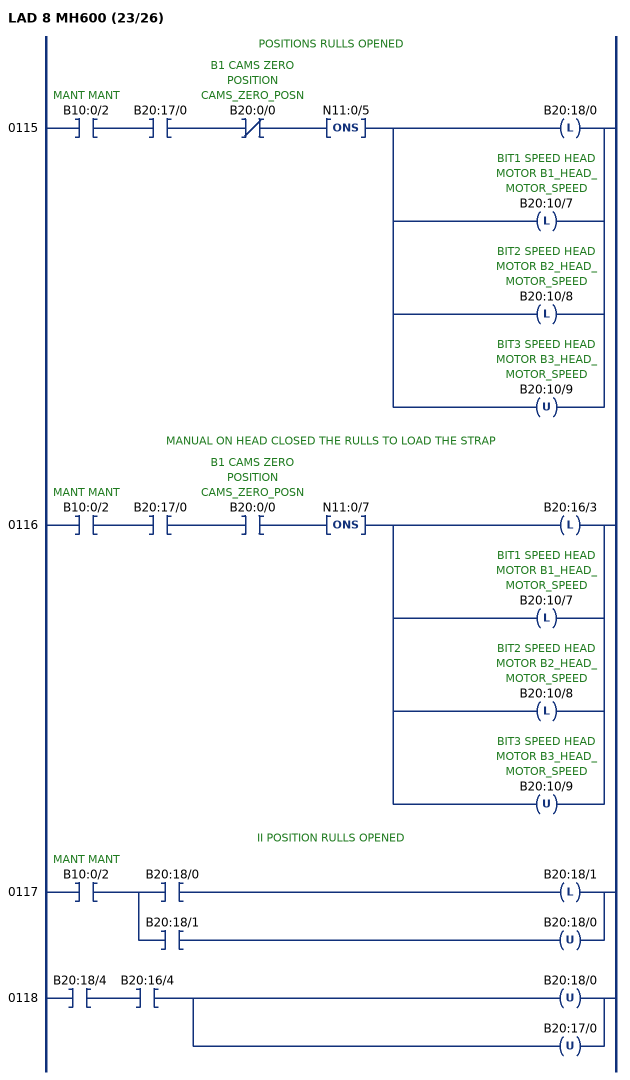
% Rung: 115 %
% POSITIONS RULLS OPENED %
SOR XIC B10:0/2 XIC B20:17/0 XIO B20:0/0 ONS N11:0/5 BST OTL B20:18/0 NXB BST OTL B20:10/7 NXB BST OTL B20:10/8 NXB OTU B20:10/9 BND BND BND EOR
%   B10:0/2  MANT  "MANT" %
%   B20:0/0  CAMS_ZERO_POSN  "B1 CAMS ZERO POSITION" %
%   B20:10/7  B1_HEAD_MOTOR_SPEED  "BIT1 SPEED HEAD MOTOR" %
%   B20:10/8  B2_HEAD_MOTOR_SPEED  "BIT2 SPEED HEAD MOTOR" %
%   B20:10/9  B3_HEAD_MOTOR_SPEED  "BIT3 SPEED HEAD MOTOR" %
% Rung: 116 %
% MANUAL ON HEAD CLOSED THE RULLS TO LOAD THE STRAP %
SOR XIC B10:0/2 XIC B20:17/0 XIC B20:0/0 ONS N11:0/7 BST OTL B20:16/3 NXB BST OTL B20:10/7 NXB BST OTL B20:10/8 NXB OTU B20:10/9 BND BND BND EOR
%   B10:0/2  MANT  "MANT" %
%   B20:0/0  CAMS_ZERO_POSN  "B1 CAMS ZERO POSITION" %
%   B20:10/7  B1_HEAD_MOTOR_SPEED  "BIT1 SPEED HEAD MOTOR" %
%   B20:10/8  B2_HEAD_MOTOR_SPEED  "BIT2 SPEED HEAD MOTOR" %
%   B20:10/9  B3_HEAD_MOTOR_SPEED  "BIT3 SPEED HEAD MOTOR" %
% Rung: 117 %
% II POSITION RULLS OPENED %
SOR XIC B10:0/2 BST XIC B20:18/0 OTL B20:18/1 NXB XIC B20:18/1 OTU B20:18/0 BND EOR
%   B10:0/2  MANT  "MANT" %
% Rung: 118 %
SOR XIC B20:18/4 XIC B20:16/4 BST OTU B20:18/0 NXB OTU B20:17/0 BND EOR

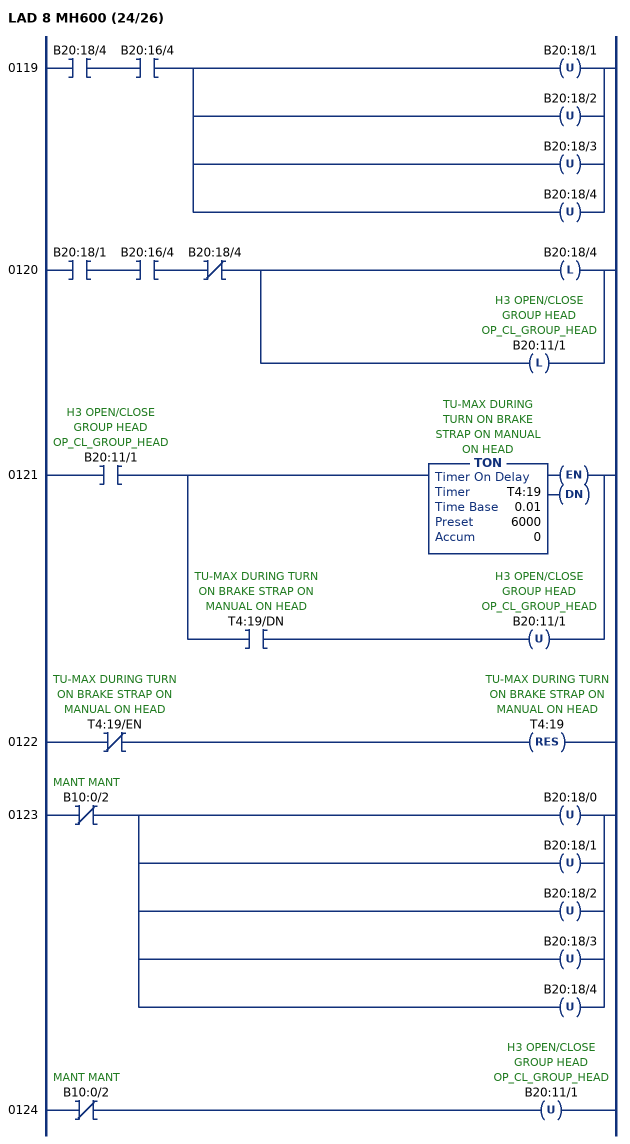
% Rung: 119 %
SOR XIC B20:18/4 XIC B20:16/4 BST OTU B20:18/1 NXB BST OTU B20:18/2 NXB BST OTU B20:18/3 NXB OTU B20:18/4 BND BND BND EOR
% Rung: 120 %
SOR XIC B20:18/1 XIC B20:16/4 XIO B20:18/4 BST OTL B20:18/4 NXB OTL B20:11/1 BND EOR
%   B20:11/1  OP_CL_GROUP_HEAD  "H3 OPEN/CLOSE GROUP HEAD" %
% Rung: 121 %
SOR XIC B20:11/1 BST TON T4:19 0.01 6000 0 NXB XIC T4:19/DN OTU B20:11/1 BND EOR
%   B20:11/1  OP_CL_GROUP_HEAD  "H3 OPEN/CLOSE GROUP HEAD" %
%   T4:19  "TU-MAX DURING TURN ON BRAKE STRAP ON MANUAL ON HEAD" %
% Rung: 122 %
SOR XIO T4:19/EN RES T4:19 EOR
%   T4:19  "TU-MAX DURING TURN ON BRAKE STRAP ON MANUAL ON HEAD" %
% Rung: 123 %
SOR XIO B10:0/2 BST OTU B20:18/0 NXB BST OTU B20:18/1 NXB BST OTU B20:18/2 NXB BST OTU B20:18/3 NXB OTU B20:18/4 BND BND BND BND EOR
%   B10:0/2  MANT  "MANT" %
% Rung: 124 %
SOR XIO B10:0/2 OTU B20:11/1 EOR
%   B10:0/2  MANT  "MANT" %
%   B20:11/1  OP_CL_GROUP_HEAD  "H3 OPEN/CLOSE GROUP HEAD" %

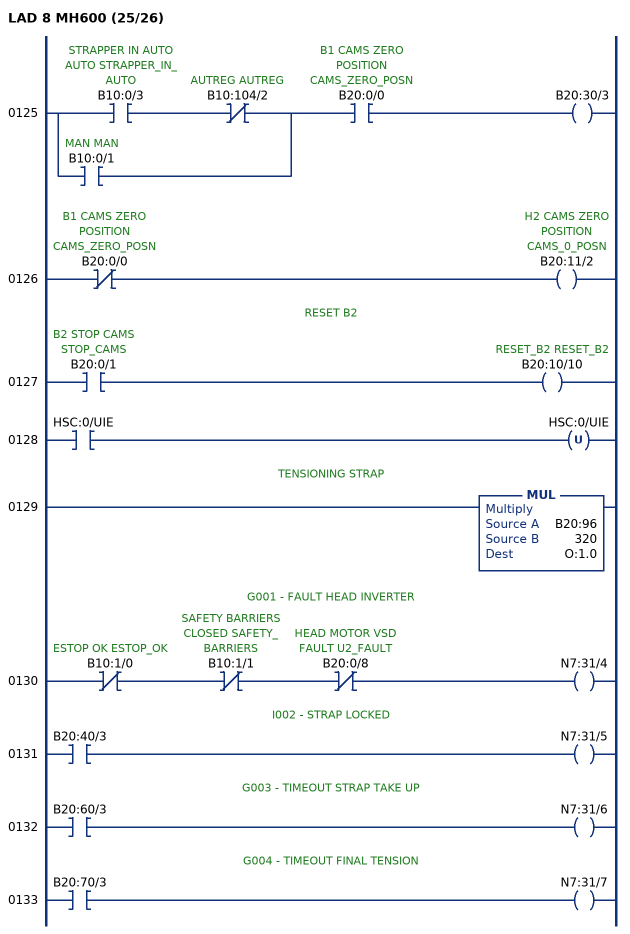
% Rung: 125 %
SOR BST XIC B10:0/3 XIO B10:104/2 NXB XIC B10:0/1 BND XIC B20:0/0 OTE B20:30/3 EOR
%   B10:0/3  STRAPPER_IN_AUTO  "STRAPPER IN AUTO AUTO" %
%   B10:104/2  AUTREG  "AUTREG" %
%   B10:0/1  MAN  "MAN" %
%   B20:0/0  CAMS_ZERO_POSN  "B1 CAMS ZERO POSITION" %
% Rung: 126 %
SOR XIO B20:0/0 OTE B20:11/2 EOR
%   B20:0/0  CAMS_ZERO_POSN  "B1 CAMS ZERO POSITION" %
%   B20:11/2  CAMS_0_POSN  "H2 CAMS ZERO POSITION" %
% Rung: 127 %
% RESET B2 %
SOR XIC B20:0/1 OTE B20:10/10 EOR
%   B20:0/1  STOP_CAMS  "B2 STOP CAMS" %
%   B20:10/10  RESET_B2  "RESET_B2" %
% Rung: 128 %
SOR XIC HSC:0/UIE OTU HSC:0/UIE EOR
% Rung: 129 %
% TENSIONING STRAP %
SOR MUL B20:96 320 O:1.0 EOR
% Rung: 130 %
% G001 - FAULT HEAD INVERTER %
SOR XIO B10:1/0 XIO B10:1/1 XIO B20:0/8 OTE N7:31/4 EOR
%   B10:1/0  ESTOP_OK  "ESTOP OK" %
%   B10:1/1  SAFETY_BARRIERS  "SAFETY BARRIERS CLOSED" %
%   B20:0/8  U2_FAULT  "HEAD MOTOR VSD FAULT" %
% Rung: 131 %
% I002 - STRAP LOCKED %
SOR XIC B20:40/3 OTE N7:31/5 EOR
% Rung: 132 %
% G003 - TIMEOUT STRAP TAKE UP %
SOR XIC B20:60/3 OTE N7:31/6 EOR
% Rung: 133 %
% G004 - TIMEOUT FINAL TENSION %
SOR XIC B20:70/3 OTE N7:31/7 EOR

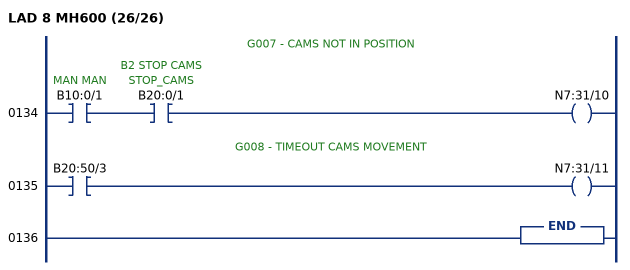
% Rung: 134 %
% G007 - CAMS NOT IN POSITION %
SOR XIC B10:0/1 XIC B20:0/1 OTE N7:31/10 EOR
%   B10:0/1  MAN  "MAN" %
%   B20:0/1  STOP_CAMS  "B2 STOP CAMS" %
% Rung: 135 %
% G008 - TIMEOUT CAMS MOVEMENT %
SOR XIC B20:50/3 OTE N7:31/11 EOR
% Rung: 136 %
SOR END EOR

LADDER 9 "ORGANIT."
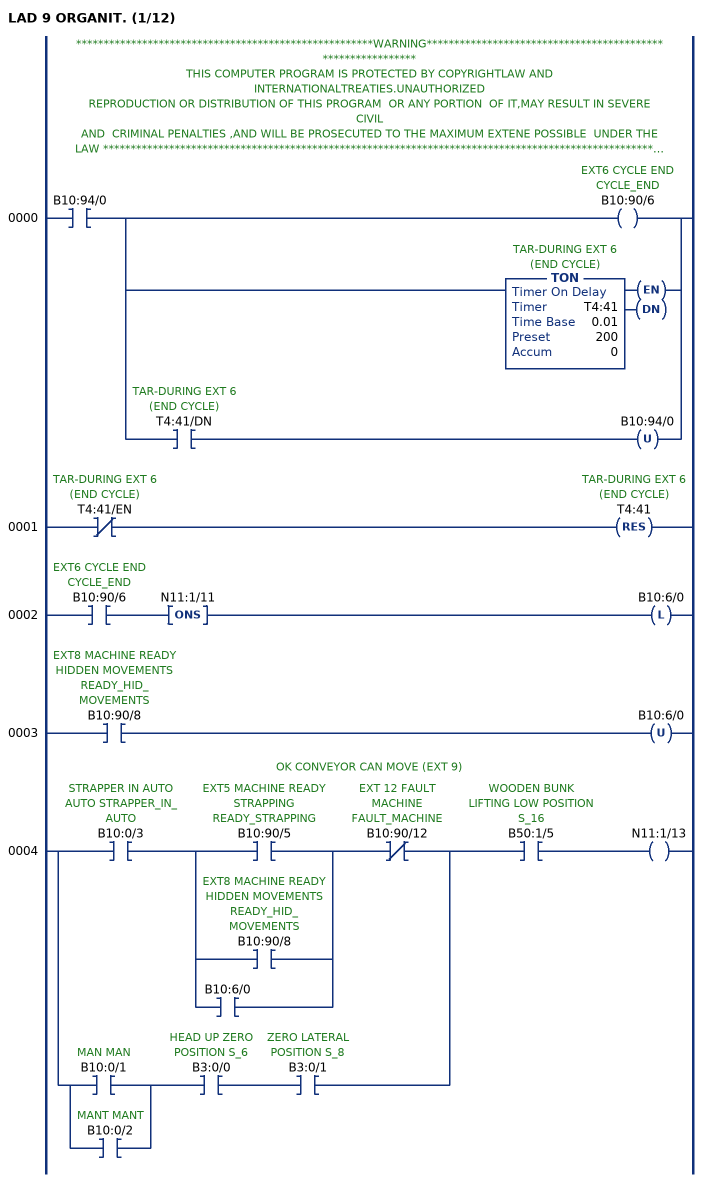
% Rung: 0 %
% ******************************************************WARNING************************************************************
% THIS COMPUTER PROGRAM IS PROTECTED BY COPYRIGHTLAW AND  INTERNATIONALTREATIES.UNAUTHORIZED
%  REPRODUCTION OR DISTRIBUTION OF THIS PROGRAM  OR ANY PORTION  OF IT,MAY RESULT IN SEVERE CIVIL
% AND  CRIMINAL PENALTIES ,AND WILL BE PROSECUTED TO THE MAXIMUM EXTENE POSSIBLE  UNDER THE LAW **************************************************************************************************************************
% INTERFACE SIGNALS - CYCLE END %
SOR XIC B10:94/0 BST OTE B10:90/6 NXB BST TON T4:41 0.01 200 0 NXB XIC T4:41/DN OTU B10:94/0 BND BND EOR
%   B10:90/6  CYCLE_END  "EXT6 CYCLE END" %
%   T4:41  "TAR-DURING EXT 6 (END CYCLE)" %
% Rung: 1 %
SOR XIO T4:41/EN RES T4:41 EOR
%   T4:41  "TAR-DURING EXT 6 (END CYCLE)" %
% Rung: 2 %
SOR XIC B10:90/6 ONS N11:1/11 OTL B10:6/0 EOR
%   B10:90/6  CYCLE_END  "EXT6 CYCLE END" %
% Rung: 3 %
SOR XIC B10:90/8 OTU B10:6/0 EOR
%   B10:90/8  READY_HID_MOVEMENTS  "EXT8 MACHINE READY HIDDEN MOVEMENTS" %
% Rung: 4 %
% OK CONVEYOR CAN MOVE (EXT 9) %
SOR BST XIC B10:0/3 BST XIC B10:90/5 NXB BST XIC B10:90/8 NXB XIC B10:6/0 BND BND XIO B10:90/12 NXB BST XIC B10:0/1 NXB XIC B10:0/2 BND XIC B3:0/0 XIC B3:0/1 BND XIC B50:1/5 OTE N11:1/13 EOR
%   B10:0/3  STRAPPER_IN_AUTO  "STRAPPER IN AUTO AUTO" %
%   B10:90/5  READY_STRAPPING  "EXT5 MACHINE READY STRAPPING" %
%   B10:90/8  READY_HID_MOVEMENTS  "EXT8 MACHINE READY HIDDEN MOVEMENTS" %
%   B10:90/12  FAULT_MACHINE  "EXT 12 FAULT MACHINE" %
%   B10:0/1  MAN  "MAN" %
%   B10:0/2  MANT  "MANT" %
%   B3:0/0  S_6  "HEAD UP ZERO POSITION" %
%   B3:0/1  S_8  "ZERO LATERAL POSITION" %
%   B50:1/5  S_16  "WOODEN BUNK LIFTING LOW POSITION" %

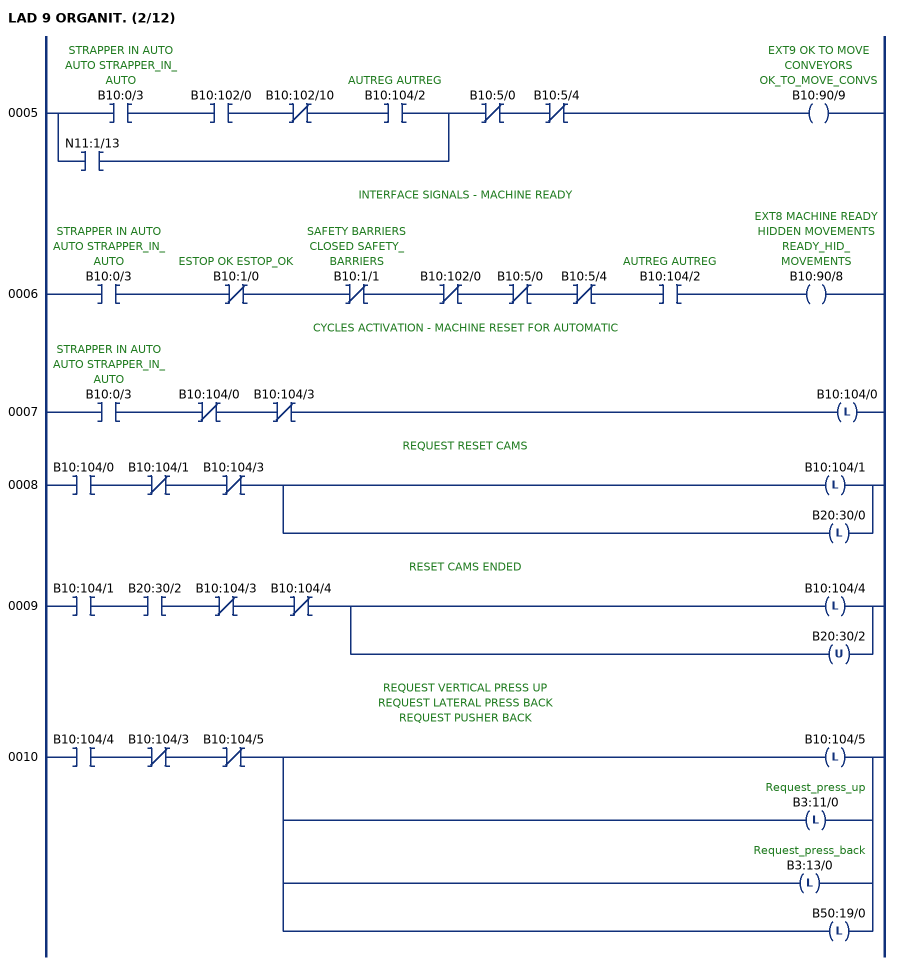
% Rung: 5 %
SOR BST XIC B10:0/3 XIC B10:102/0 XIO B10:102/10 XIC B10:104/2 NXB XIC N11:1/13 BND XIO B10:5/0 XIO B10:5/4 OTE B10:90/9 EOR
%   B10:0/3  STRAPPER_IN_AUTO  "STRAPPER IN AUTO AUTO" %
%   B10:104/2  AUTREG  "AUTREG" %
%   B10:90/9  OK_TO_MOVE_CONVS  "EXT9 OK TO MOVE CONVEYORS" %
% Rung: 6 %
% INTERFACE SIGNALS - MACHINE READY %
SOR XIC B10:0/3 XIO B10:1/0 XIO B10:1/1 XIO B10:102/0 XIO B10:5/0 XIO B10:5/4 XIC B10:104/2 OTE B10:90/8 EOR
%   B10:0/3  STRAPPER_IN_AUTO  "STRAPPER IN AUTO AUTO" %
%   B10:1/0  ESTOP_OK  "ESTOP OK" %
%   B10:1/1  SAFETY_BARRIERS  "SAFETY BARRIERS CLOSED" %
%   B10:104/2  AUTREG  "AUTREG" %
%   B10:90/8  READY_HID_MOVEMENTS  "EXT8 MACHINE READY HIDDEN MOVEMENTS" %
% Rung: 7 %
% CYCLES ACTIVATION - MACHINE RESET FOR AUTOMATIC %
SOR XIC B10:0/3 XIO B10:104/0 XIO B10:104/3 OTL B10:104/0 EOR
%   B10:0/3  STRAPPER_IN_AUTO  "STRAPPER IN AUTO AUTO" %
% Rung: 8 %
% REQUEST RESET CAMS %
SOR XIC B10:104/0 XIO B10:104/1 XIO B10:104/3 BST OTL B10:104/1 NXB OTL B20:30/0 BND EOR
% Rung: 9 %
% RESET CAMS ENDED %
SOR XIC B10:104/1 XIC B20:30/2 XIO B10:104/3 XIO B10:104/4 BST OTL B10:104/4 NXB OTU B20:30/2 BND EOR
% Rung: 10 %
% REQUEST VERTICAL PRESS UP
% REQUEST LATERAL PRESS BACK
% REQUEST PUSHER BACK %
SOR XIC B10:104/4 XIO B10:104/3 XIO B10:104/5 BST OTL B10:104/5 NXB BST OTL B3:11/0 NXB BST OTL B3:13/0 NXB OTL B50:19/0 BND BND BND EOR
%   B3:11/0  "Request_press_up" %
%   B3:13/0  "Request_press_back" %

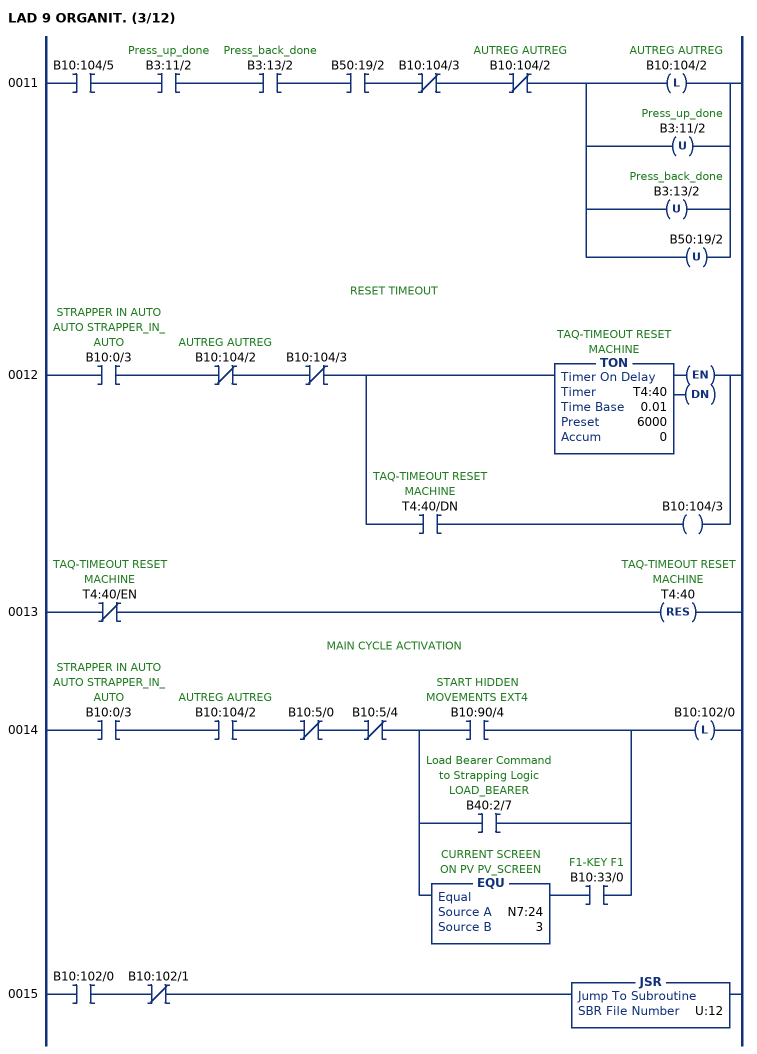
% Rung: 11 %
SOR XIC B10:104/5 XIC B3:11/2 XIC B3:13/2 XIC B50:19/2 XIO B10:104/3 XIO B10:104/2 BST OTL B10:104/2 NXB BST BST OTU B3:11/2 NXB OTU B3:13/2 BND NXB OTU B50:19/2 BND BND EOR
%   B3:11/2  "Press_up_done" %
%   B3:13/2  "Press_back_done" %
%   B10:104/2  AUTREG  "AUTREG" %
% Rung: 12 %
% RESET TIMEOUT %
SOR XIC B10:0/3 XIO B10:104/2 XIO B10:104/3 BST TON T4:40 0.01 6000 0 NXB XIC T4:40/DN OTE B10:104/3 BND EOR
%   B10:0/3  STRAPPER_IN_AUTO  "STRAPPER IN AUTO AUTO" %
%   B10:104/2  AUTREG  "AUTREG" %
%   T4:40  "TAQ-TIMEOUT RESET MACHINE" %
% Rung: 13 %
SOR XIO T4:40/EN RES T4:40 EOR
%   T4:40  "TAQ-TIMEOUT RESET MACHINE" %
% Rung: 14 %
% MAIN CYCLE ACTIVATION %
SOR XIC B10:0/3 XIC B10:104/2 XIO B10:5/0 XIO B10:5/4 BST XIC B10:90/4 NXB XIC B40:2/7 NXB EQU N7:24 3 XIC B10:33/0 BND OTL B10:102/0 EOR
%   B10:0/3  STRAPPER_IN_AUTO  "STRAPPER IN AUTO AUTO" %
%   B10:104/2  AUTREG  "AUTREG" %
%   B10:90/4  EXT4  "START HIDDEN MOVEMENTS" %
%   B40:2/7  LOAD_BEARER  "Load Bearer Command to Strapping Logic" %
%   N7:24  PV_SCREEN  "CURRENT SCREEN ON PV" %
%   B10:33/0  F1  "F1-KEY" %
% Rung: 15 %
SOR XIC B10:102/0 XIO B10:102/1 JSR U:12 EOR

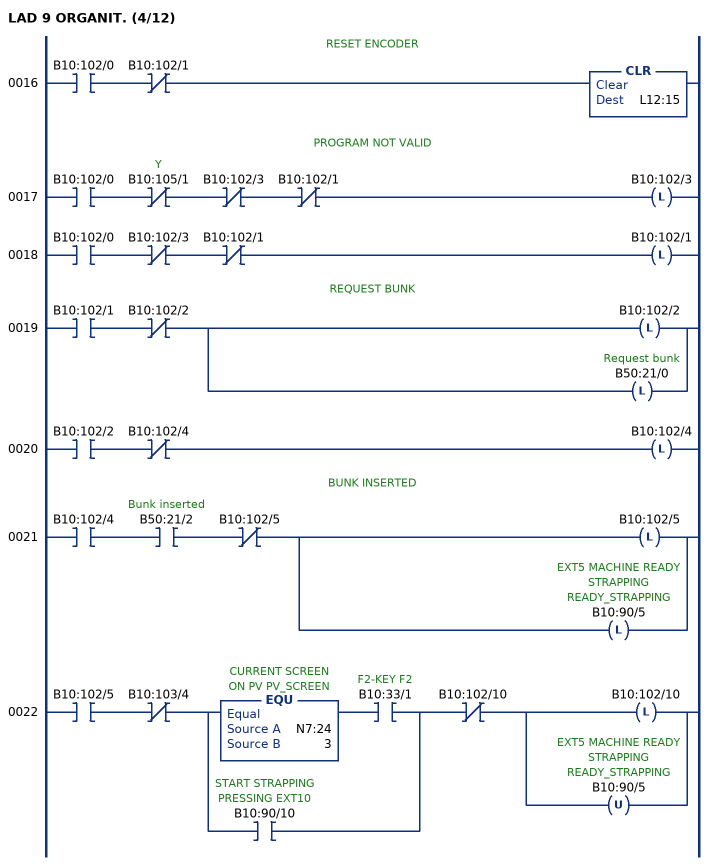
% Rung: 16 %
% RESET ENCODER %
SOR XIC B10:102/0 XIO B10:102/1 CLR L12:15 EOR
% Rung: 17 %
% PROGRAM NOT VALID %
SOR XIC B10:102/0 XIO B10:105/1 XIO B10:102/3 XIO B10:102/1 OTL B10:102/3 EOR
%   B10:105/1  "Y" %
% Rung: 18 %
SOR XIC B10:102/0 XIO B10:102/3 XIO B10:102/1 OTL B10:102/1 EOR
% Rung: 19 %
% REQUEST BUNK %
SOR XIC B10:102/1 XIO B10:102/2 BST OTL B10:102/2 NXB OTL B50:21/0 BND EOR
%   B50:21/0  "Request bunk" %
% Rung: 20 %
SOR XIC B10:102/2 XIO B10:102/4 OTL B10:102/4 EOR
% Rung: 21 %
% BUNK INSERTED %
SOR XIC B10:102/4 XIC B50:21/2 XIO B10:102/5 BST OTL B10:102/5 NXB OTL B10:90/5 BND EOR
%   B50:21/2  "Bunk inserted" %
%   B10:90/5  READY_STRAPPING  "EXT5 MACHINE READY STRAPPING" %
% Rung: 22 %
SOR XIC B10:102/5 XIO B10:103/4 BST EQU N7:24 3 XIC B10:33/1 NXB XIC B10:90/10 BND XIO B10:102/10 BST OTL B10:102/10 NXB OTU B10:90/5 BND EOR
%   N7:24  PV_SCREEN  "CURRENT SCREEN ON PV" %
%   B10:33/1  F2  "F2-KEY" %
%   B10:90/10  EXT10  "START STRAPPING PRESSING" %
%   B10:90/5  READY_STRAPPING  "EXT5 MACHINE READY STRAPPING" %

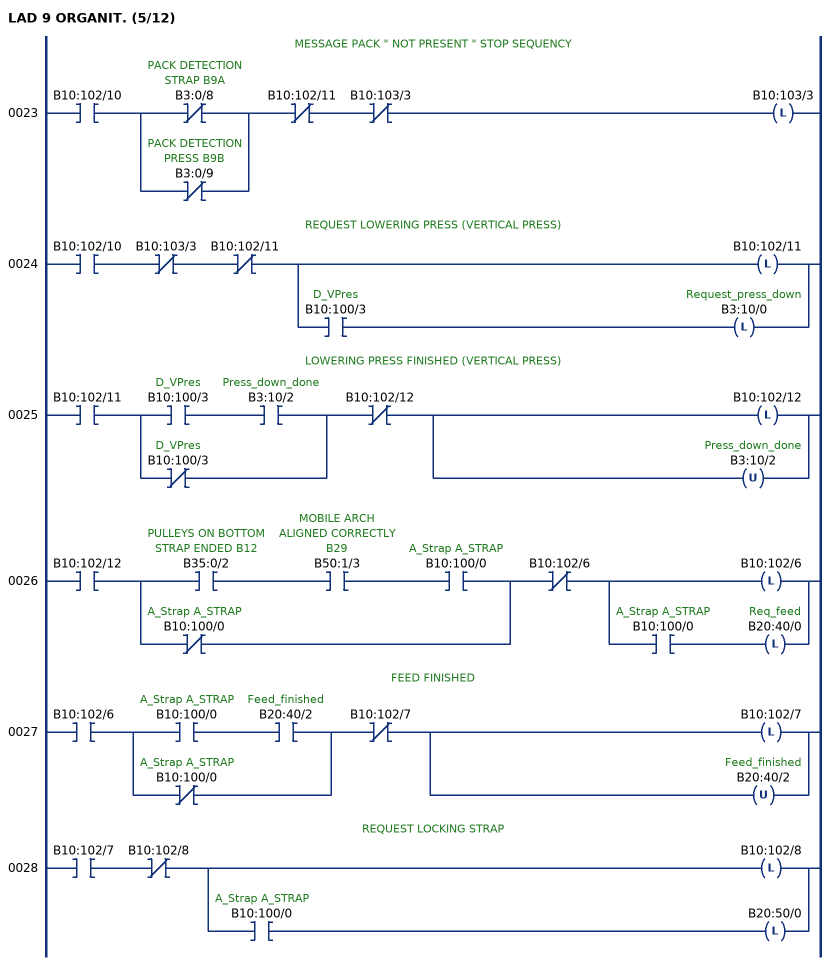
% Rung: 23 %
% MESSAGE PACK " NOT PRESENT " STOP SEQUENCY %
SOR XIC B10:102/10 BST XIO B3:0/8 NXB XIO B3:0/9 BND XIO B10:102/11 XIO B10:103/3 OTL B10:103/3 EOR
%   B3:0/8  B9A  "PACK DETECTION STRAP" %
%   B3:0/9  B9B  "PACK DETECTION PRESS" %
% Rung: 24 %
% REQUEST LOWERING PRESS (VERTICAL PRESS) %
SOR XIC B10:102/10 XIO B10:103/3 XIO B10:102/11 BST OTL B10:102/11 NXB XIC B10:100/3 OTL B3:10/0 BND EOR
%   B10:100/3  "D_VPres" %
%   B3:10/0  "Request_press_down" %
% Rung: 25 %
% LOWERING PRESS FINISHED (VERTICAL PRESS) %
SOR XIC B10:102/11 BST XIC B10:100/3 XIC B3:10/2 NXB XIO B10:100/3 BND XIO B10:102/12 BST OTL B10:102/12 NXB OTU B3:10/2 BND EOR
%   B10:100/3  "D_VPres" %
%   B3:10/2  "Press_down_done" %
% Rung: 26 %
SOR XIC B10:102/12 BST XIC B35:0/2 XIC B50:1/3 XIC B10:100/0 NXB XIO B10:100/0 BND XIO B10:102/6 BST OTL B10:102/6 NXB XIC B10:100/0 OTL B20:40/0 BND EOR
%   B35:0/2  B12  "PULLEYS ON BOTTOM STRAP ENDED" %
%   B50:1/3  B29  "MOBILE ARCH ALIGNED CORRECTLY" %
%   B10:100/0  A_STRAP  "A_Strap" %
%   B20:40/0  "Req_feed" %
% Rung: 27 %
% FEED FINISHED %
SOR XIC B10:102/6 BST XIC B10:100/0 XIC B20:40/2 NXB XIO B10:100/0 BND XIO B10:102/7 BST OTL B10:102/7 NXB OTU B20:40/2 BND EOR
%   B10:100/0  A_STRAP  "A_Strap" %
%   B20:40/2  "Feed_finished" %
% Rung: 28 %
% REQUEST LOCKING STRAP %
SOR XIC B10:102/7 XIO B10:102/8 BST OTL B10:102/8 NXB XIC B10:100/0 OTL B20:50/0 BND EOR
%   B10:100/0  A_STRAP  "A_Strap" %

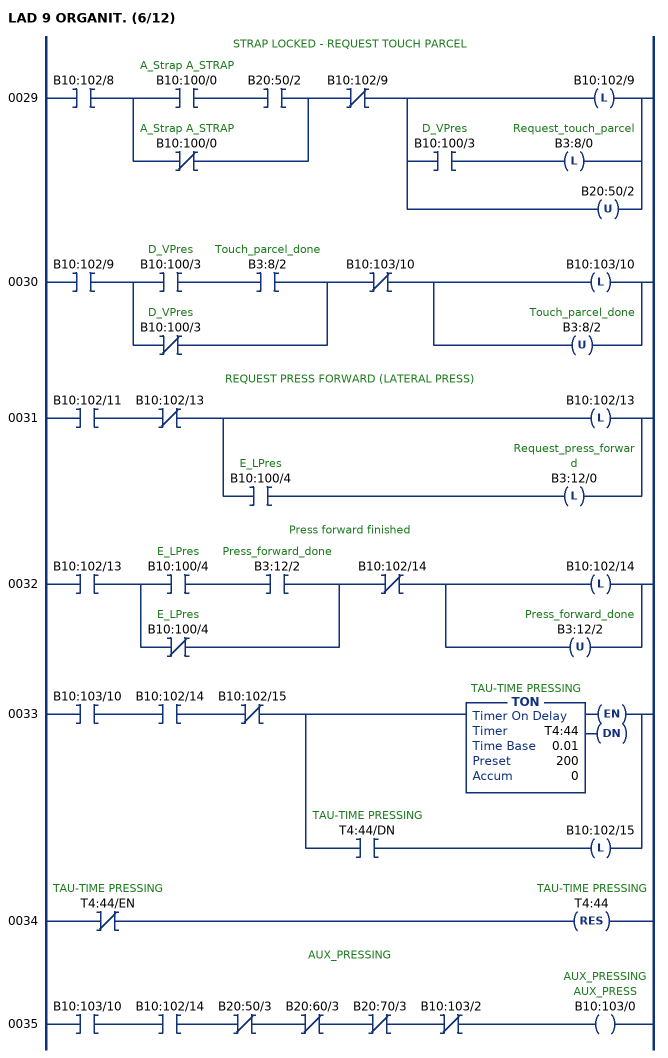
% Rung: 29 %
% STRAP LOCKED - REQUEST TOUCH PARCEL %
SOR XIC B10:102/8 BST XIC B10:100/0 XIC B20:50/2 NXB XIO B10:100/0 BND XIO B10:102/9 BST BST OTL B10:102/9 NXB XIC B10:100/3 OTL B3:8/0 BND NXB OTU B20:50/2 BND EOR
%   B10:100/0  A_STRAP  "A_Strap" %
%   B10:100/3  "D_VPres" %
%   B3:8/0  "Request_touch_parcel" %
% Rung: 30 %
SOR XIC B10:102/9 BST XIC B10:100/3 XIC B3:8/2 NXB XIO B10:100/3 BND XIO B10:103/10 BST OTL B10:103/10 NXB OTU B3:8/2 BND EOR
%   B10:100/3  "D_VPres" %
%   B3:8/2  "Touch_parcel_done" %
% Rung: 31 %
% REQUEST PRESS FORWARD (LATERAL PRESS) %
SOR XIC B10:102/11 XIO B10:102/13 BST OTL B10:102/13 NXB XIC B10:100/4 OTL B3:12/0 BND EOR
%   B10:100/4  "E_LPres" %
%   B3:12/0  "Request_press_forwar d" %
% Rung: 32 %
% Press forward finished %
SOR XIC B10:102/13 BST XIC B10:100/4 XIC B3:12/2 NXB XIO B10:100/4 BND XIO B10:102/14 BST OTL B10:102/14 NXB OTU B3:12/2 BND EOR
%   B10:100/4  "E_LPres" %
%   B3:12/2  "Press_forward_done" %
% Rung: 33 %
SOR XIC B10:103/10 XIC B10:102/14 XIO B10:102/15 BST TON T4:44 0.01 200 0 NXB XIC T4:44/DN OTL B10:102/15 BND EOR
%   T4:44  "TAU-TIME PRESSING" %
% Rung: 34 %
SOR XIO T4:44/EN RES T4:44 EOR
%   T4:44  "TAU-TIME PRESSING" %
% Rung: 35 %
% AUX_PRESSING %
SOR XIC B10:103/10 XIC B10:102/14 XIO B20:50/3 XIO B20:60/3 XIO B20:70/3 XIO B10:103/2 OTE B10:103/0 EOR
%   B10:103/0  AUX_PRESS  "AUX_PRESSING" %

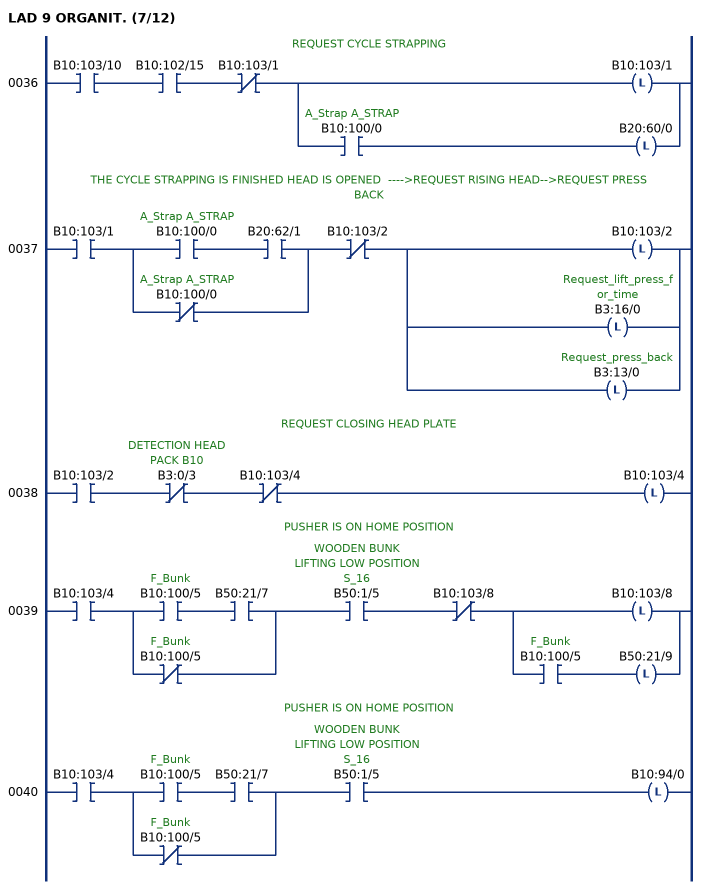
% Rung: 36 %
% REQUEST CYCLE STRAPPING %
SOR XIC B10:103/10 XIC B10:102/15 XIO B10:103/1 BST OTL B10:103/1 NXB XIC B10:100/0 OTL B20:60/0 BND EOR
%   B10:100/0  A_STRAP  "A_Strap" %
% Rung: 37 %
% THE CYCLE STRAPPING IS FINISHED HEAD IS OPENED  ---->REQUEST RISING HEAD-->REQUEST PRESS BACK %
SOR XIC B10:103/1 BST XIC B10:100/0 XIC B20:62/1 NXB XIO B10:100/0 BND XIO B10:103/2 BST OTL B10:103/2 NXB BST OTL B3:16/0 NXB OTL B3:13/0 BND BND EOR
%   B10:100/0  A_STRAP  "A_Strap" %
%   B3:16/0  "Request_lift_press_f or_time" %
%   B3:13/0  "Request_press_back" %
% Rung: 38 %
% REQUEST CLOSING HEAD PLATE %
SOR XIC B10:103/2 XIO B3:0/3 XIO B10:103/4 OTL B10:103/4 EOR
%   B3:0/3  B10  "DETECTION HEAD PACK" %
% Rung: 39 %
% PUSHER IS ON HOME POSITION %
SOR XIC B10:103/4 BST XIC B10:100/5 XIC B50:21/7 NXB XIO B10:100/5 BND XIC B50:1/5 XIO B10:103/8 BST OTL B10:103/8 NXB XIC B10:100/5 OTL B50:21/9 BND EOR
%   B10:100/5  "F_Bunk" %
%   B50:1/5  S_16  "WOODEN BUNK LIFTING LOW POSITION" %
% Rung: 40 %
% PUSHER IS ON HOME POSITION %
SOR XIC B10:103/4 BST XIC B10:100/5 XIC B50:21/7 NXB XIO B10:100/5 BND XIC B50:1/5 OTL B10:94/0 EOR
%   B10:100/5  "F_Bunk" %
%   B50:1/5  S_16  "WOODEN BUNK LIFTING LOW POSITION" %

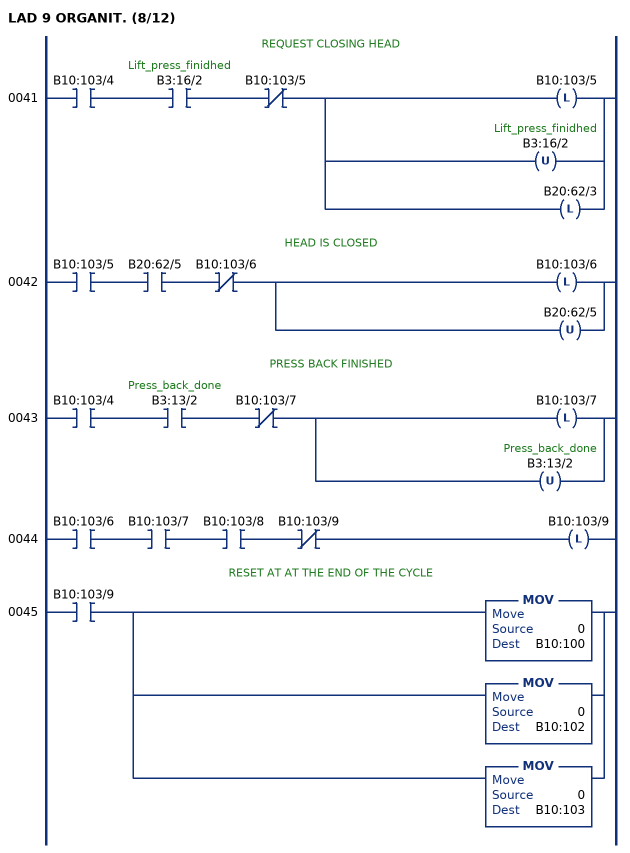
% Rung: 41 %
% REQUEST CLOSING HEAD %
SOR XIC B10:103/4 XIC B3:16/2 XIO B10:103/5 BST BST OTL B10:103/5 NXB OTU B3:16/2 BND NXB OTL B20:62/3 BND EOR
%   B3:16/2  "Lift_press_finidhed" %
% Rung: 42 %
% HEAD IS CLOSED %
SOR XIC B10:103/5 XIC B20:62/5 XIO B10:103/6 BST OTL B10:103/6 NXB OTU B20:62/5 BND EOR
% Rung: 43 %
% PRESS BACK FINISHED %
SOR XIC B10:103/4 XIC B3:13/2 XIO B10:103/7 BST OTL B10:103/7 NXB OTU B3:13/2 BND EOR
%   B3:13/2  "Press_back_done" %
% Rung: 44 %
SOR XIC B10:103/6 XIC B10:103/7 XIC B10:103/8 XIO B10:103/9 OTL B10:103/9 EOR
% Rung: 45 %
% RESET AT AT THE END OF THE CYCLE %
SOR XIC B10:103/9 BST MOV 0 B10:100 NXB BST MOV 0 B10:102 NXB MOV 0 B10:103 BND BND EOR

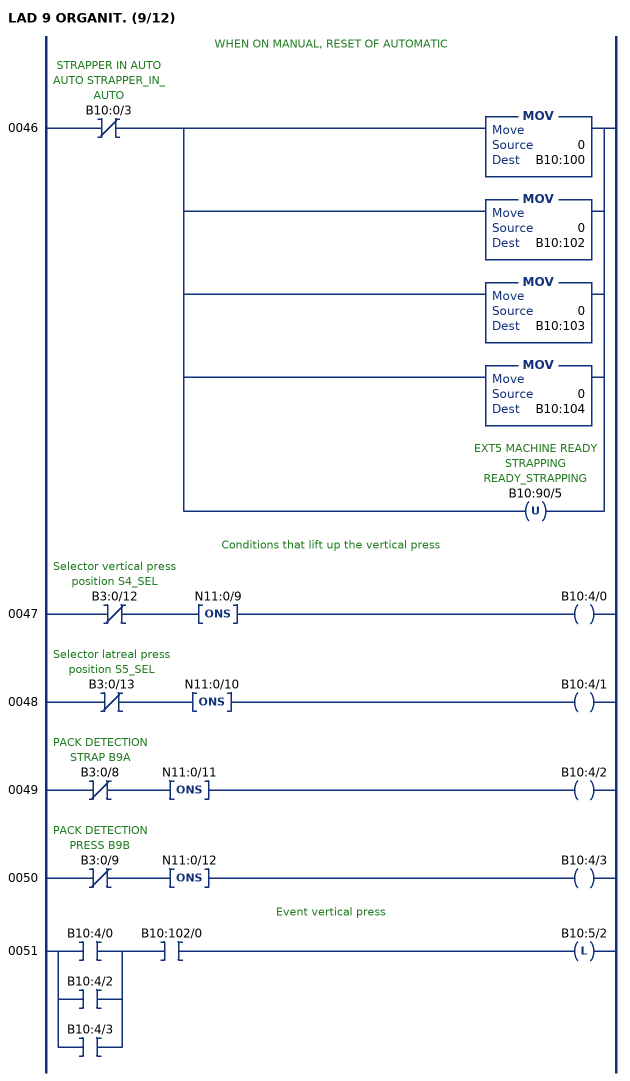
% Rung: 46 %
% WHEN ON MANUAL, RESET OF AUTOMATIC %
SOR XIO B10:0/3 BST MOV 0 B10:100 NXB BST BST MOV 0 B10:102 NXB MOV 0 B10:103 BND NXB BST MOV 0 B10:104 NXB OTU B10:90/5 BND BND BND EOR
%   B10:0/3  STRAPPER_IN_AUTO  "STRAPPER IN AUTO AUTO" %
%   B10:90/5  READY_STRAPPING  "EXT5 MACHINE READY STRAPPING" %
% Rung: 47 %
% Conditions that lift up the vertical press %
SOR XIO B3:0/12 ONS N11:0/9 OTE B10:4/0 EOR
%   B3:0/12  S4_SEL  "Selector vertical press position" %
% Rung: 48 %
SOR XIO B3:0/13 ONS N11:0/10 OTE B10:4/1 EOR
%   B3:0/13  S5_SEL  "Selector latreal press position" %
% Rung: 49 %
SOR XIO B3:0/8 ONS N11:0/11 OTE B10:4/2 EOR
%   B3:0/8  B9A  "PACK DETECTION STRAP" %
% Rung: 50 %
SOR XIO B3:0/9 ONS N11:0/12 OTE B10:4/3 EOR
%   B3:0/9  B9B  "PACK DETECTION PRESS" %
% Rung: 51 %
% Event vertical press %
SOR BST XIC B10:4/0 NXB BST XIC B10:4/2 NXB XIC B10:4/3 BND BND XIC B10:102/0 OTL B10:5/2 EOR

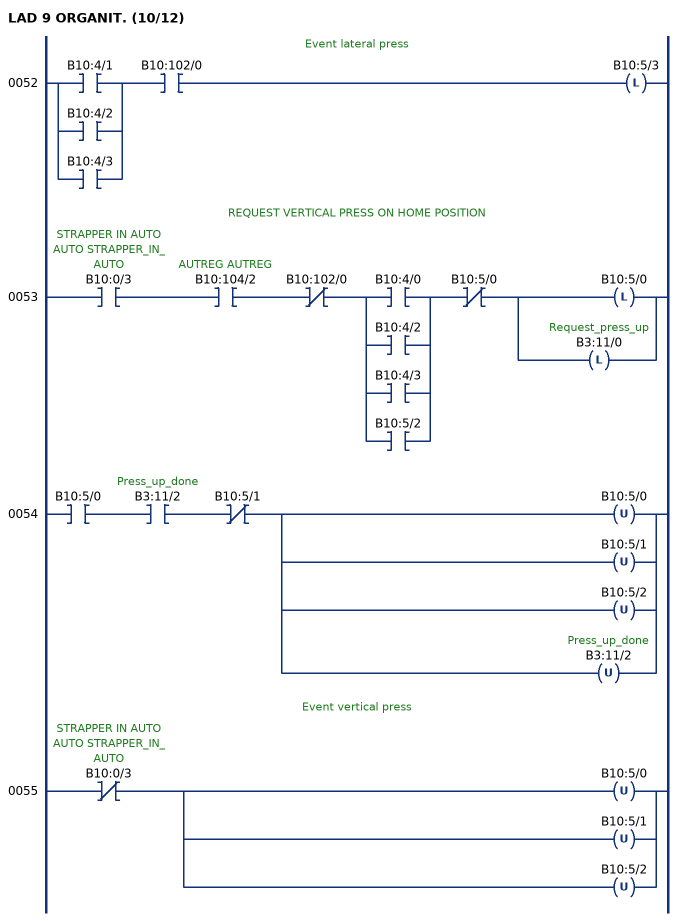
% Rung: 52 %
% Event lateral press %
SOR BST XIC B10:4/1 NXB BST XIC B10:4/2 NXB XIC B10:4/3 BND BND XIC B10:102/0 OTL B10:5/3 EOR
% Rung: 53 %
% REQUEST VERTICAL PRESS ON HOME POSITION %
SOR XIC B10:0/3 XIC B10:104/2 XIO B10:102/0 BST BST XIC B10:4/0 NXB XIC B10:4/2 BND NXB BST XIC B10:4/3 NXB XIC B10:5/2 BND BND XIO B10:5/0 BST OTL B10:5/0 NXB OTL B3:11/0 BND EOR
%   B10:0/3  STRAPPER_IN_AUTO  "STRAPPER IN AUTO AUTO" %
%   B10:104/2  AUTREG  "AUTREG" %
%   B3:11/0  "Request_press_up" %
% Rung: 54 %
SOR XIC B10:5/0 XIC B3:11/2 XIO B10:5/1 BST BST OTU B10:5/0 NXB BST OTU B10:5/1 NXB OTU B10:5/2 BND BND NXB OTU B3:11/2 BND EOR
%   B3:11/2  "Press_up_done" %
% Rung: 55 %
% Event vertical press %
SOR XIO B10:0/3 BST OTU B10:5/0 NXB BST OTU B10:5/1 NXB OTU B10:5/2 BND BND EOR
%   B10:0/3  STRAPPER_IN_AUTO  "STRAPPER IN AUTO AUTO" %

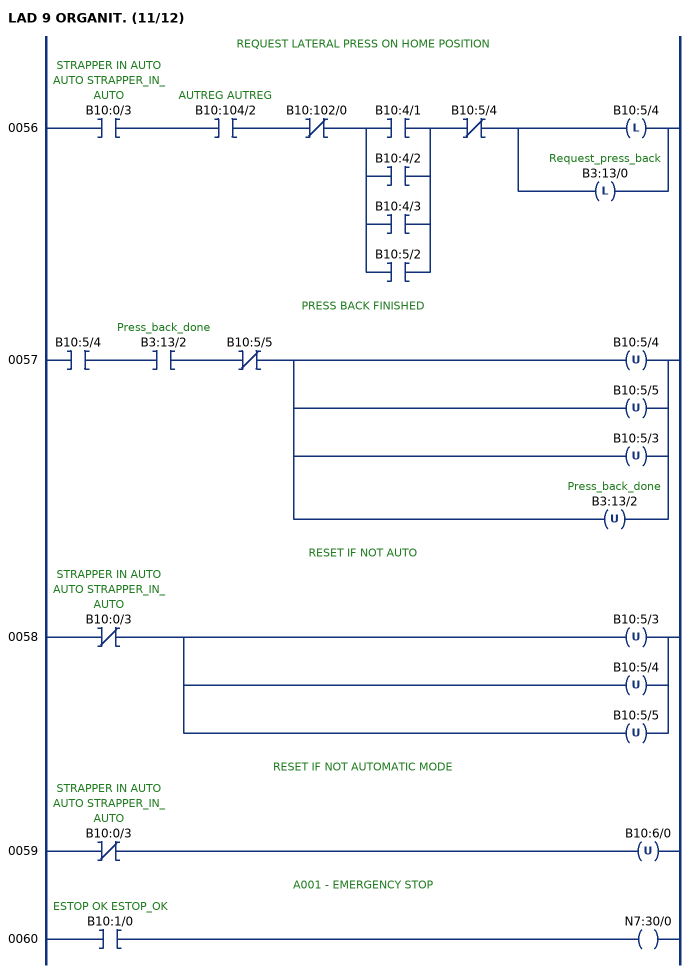
% Rung: 56 %
% REQUEST LATERAL PRESS ON HOME POSITION %
SOR XIC B10:0/3 XIC B10:104/2 XIO B10:102/0 BST BST XIC B10:4/1 NXB BST XIC B10:4/2 NXB XIC B10:4/3 BND BND NXB XIC B10:5/2 BND XIO B10:5/4 BST OTL B10:5/4 NXB OTL B3:13/0 BND EOR
%   B10:0/3  STRAPPER_IN_AUTO  "STRAPPER IN AUTO AUTO" %
%   B10:104/2  AUTREG  "AUTREG" %
%   B3:13/0  "Request_press_back" %
% Rung: 57 %
% PRESS BACK FINISHED %
SOR XIC B10:5/4 XIC B3:13/2 XIO B10:5/5 BST BST OTU B10:5/4 NXB BST OTU B10:5/5 NXB OTU B10:5/3 BND BND NXB OTU B3:13/2 BND EOR
%   B3:13/2  "Press_back_done" %
% Rung: 58 %
% RESET IF NOT AUTO %
SOR XIO B10:0/3 BST OTU B10:5/3 NXB BST OTU B10:5/4 NXB OTU B10:5/5 BND BND EOR
%   B10:0/3  STRAPPER_IN_AUTO  "STRAPPER IN AUTO AUTO" %
% Rung: 59 %
% RESET IF NOT AUTOMATIC MODE %
SOR XIO B10:0/3 OTU B10:6/0 EOR
%   B10:0/3  STRAPPER_IN_AUTO  "STRAPPER IN AUTO AUTO" %
% Rung: 60 %
% A001 - EMERGENCY STOP %
SOR XIC B10:1/0 OTE N7:30/0 EOR
%   B10:1/0  ESTOP_OK  "ESTOP OK" %

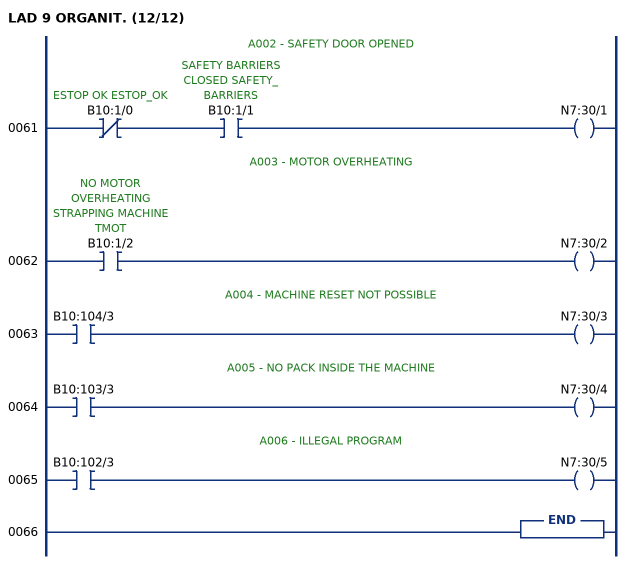
% Rung: 61 %
% A002 - SAFETY DOOR OPENED %
SOR XIO B10:1/0 XIC B10:1/1 OTE N7:30/1 EOR
%   B10:1/0  ESTOP_OK  "ESTOP OK" %
%   B10:1/1  SAFETY_BARRIERS  "SAFETY BARRIERS CLOSED" %
% Rung: 62 %
% A003 - MOTOR OVERHEATING %
SOR XIC B10:1/2 OTE N7:30/2 EOR
%   B10:1/2  TMOT  "NO MOTOR OVERHEATING STRAPPING MACHINE" %
% Rung: 63 %
% A004 - MACHINE RESET NOT POSSIBLE %
SOR XIC B10:104/3 OTE N7:30/3 EOR
% Rung: 64 %
% A005 - NO PACK INSIDE THE MACHINE %
SOR XIC B10:103/3 OTE N7:30/4 EOR
% Rung: 65 %
% A006 - ILLEGAL PROGRAM %
SOR XIC B10:102/3 OTE N7:30/5 EOR
% Rung: 66 %
SOR END EOR

LADDER 10 "PRESS"
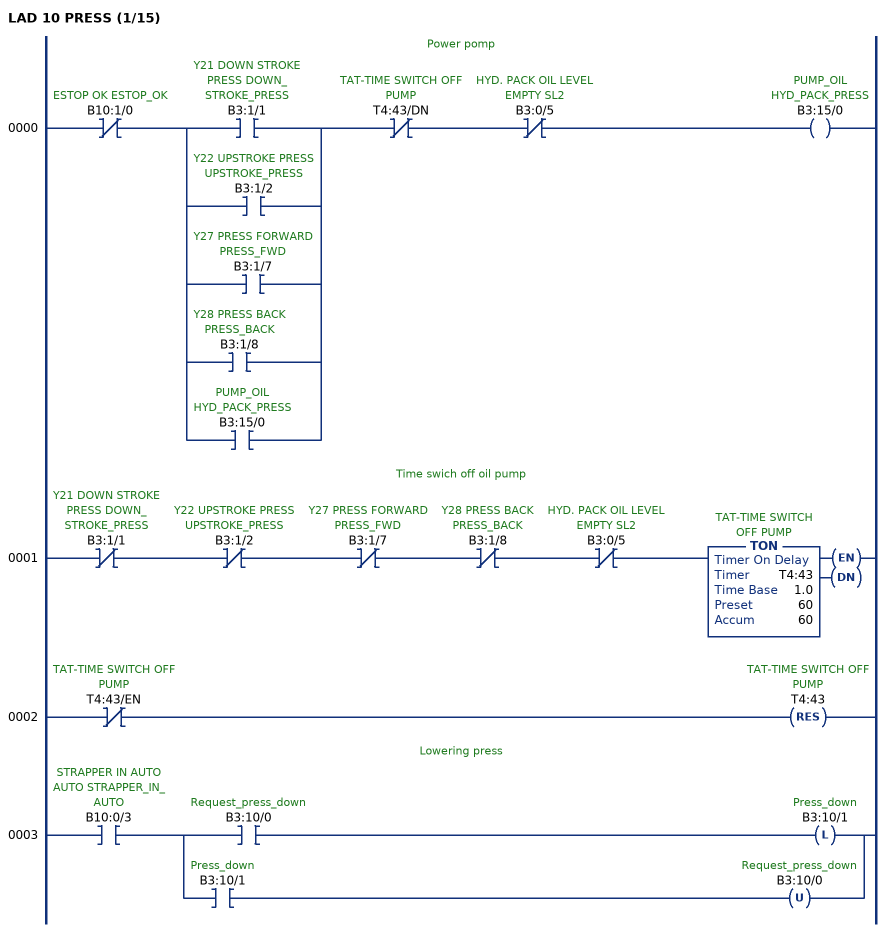
% Rung: 0 %
% Power pomp %
SOR XIO B10:1/0 BST BST XIC B3:1/1 NXB BST XIC B3:1/2 NXB BST XIC B3:1/7 NXB XIC B3:1/8 BND BND BND NXB XIC B3:15/0 BND XIO T4:43/DN XIO B3:0/5 OTE B3:15/0 EOR
%   B10:1/0  ESTOP_OK  "ESTOP OK" %
%   B3:1/1  DOWN_STROKE_PRESS  "Y21 DOWN STROKE PRESS" %
%   B3:1/2  UPSTROKE_PRESS  "Y22 UPSTROKE PRESS" %
%   B3:1/7  PRESS_FWD  "Y27 PRESS FORWARD" %
%   B3:1/8  PRESS_BACK  "Y28 PRESS BACK" %
%   B3:15/0  HYD_PACK_PRESS  "PUMP_OIL" %
%   T4:43  "TAT-TIME SWITCH OFF PUMP" %
%   B3:0/5  SL2  "HYD. PACK OIL LEVEL EMPTY" %
% Rung: 1 %
% Time swich off oil pump %
SOR XIO B3:1/1 XIO B3:1/2 XIO B3:1/7 XIO B3:1/8 XIO B3:0/5 TON T4:43 1.0 60 60 EOR
%   B3:1/1  DOWN_STROKE_PRESS  "Y21 DOWN STROKE PRESS" %
%   B3:1/2  UPSTROKE_PRESS  "Y22 UPSTROKE PRESS" %
%   B3:1/7  PRESS_FWD  "Y27 PRESS FORWARD" %
%   B3:1/8  PRESS_BACK  "Y28 PRESS BACK" %
%   B3:0/5  SL2  "HYD. PACK OIL LEVEL EMPTY" %
%   T4:43  "TAT-TIME SWITCH OFF PUMP" %
% Rung: 2 %
SOR XIO T4:43/EN RES T4:43 EOR
%   T4:43  "TAT-TIME SWITCH OFF PUMP" %
% Rung: 3 %
% Lowering press %
SOR XIC B10:0/3 BST XIC B3:10/0 OTL B3:10/1 NXB XIC B3:10/1 OTU B3:10/0 BND EOR
%   B10:0/3  STRAPPER_IN_AUTO  "STRAPPER IN AUTO AUTO" %
%   B3:10/0  "Request_press_down" %
%   B3:10/1  "Press_down" %

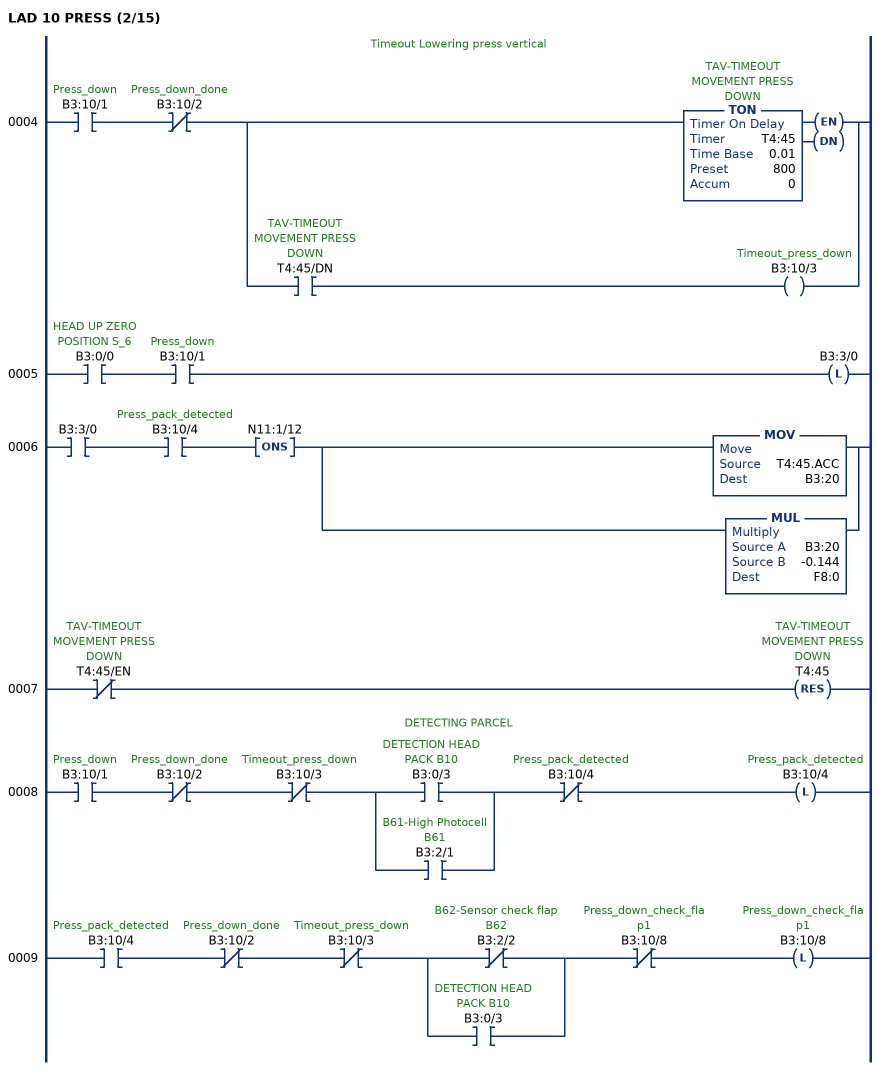
% Rung: 4 %
% Timeout Lowering press vertical %
SOR XIC B3:10/1 XIO B3:10/2 BST TON T4:45 0.01 800 0 NXB XIC T4:45/DN OTE B3:10/3 BND EOR
%   B3:10/1  "Press_down" %
%   B3:10/2  "Press_down_done" %
%   T4:45  "TAV-TIMEOUT MOVEMENT PRESS DOWN" %
%   B3:10/3  "Timeout_press_down" %
% Rung: 5 %
SOR XIC B3:0/0 XIC B3:10/1 OTL B3:3/0 EOR
%   B3:0/0  S_6  "HEAD UP ZERO POSITION" %
%   B3:10/1  "Press_down" %
% Rung: 6 %
SOR XIC B3:3/0 XIC B3:10/4 ONS N11:1/12 BST MOV T4:45.ACC B3:20 NXB MUL B3:20 -0.144 F8:0 BND EOR
%   B3:10/4  "Press_pack_detected" %
%   T4:45  "TAV-TIMEOUT MOVEMENT PRESS DOWN" %
% Rung: 7 %
SOR XIO T4:45/EN RES T4:45 EOR
%   T4:45  "TAV-TIMEOUT MOVEMENT PRESS DOWN" %
% Rung: 8 %
% DETECTING PARCEL %
SOR XIC B3:10/1 XIO B3:10/2 XIO B3:10/3 BST XIC B3:0/3 NXB XIC B3:2/1 BND XIO B3:10/4 OTL B3:10/4 EOR
%   B3:10/1  "Press_down" %
%   B3:10/2  "Press_down_done" %
%   B3:10/3  "Timeout_press_down" %
%   B3:0/3  B10  "DETECTION HEAD PACK" %
%   B3:2/1  B61  "B61-High Photocell" %
%   B3:10/4  "Press_pack_detected" %
% Rung: 9 %
SOR XIC B3:10/4 XIO B3:10/2 XIO B3:10/3 BST XIO B3:2/2 NXB XIC B3:0/3 BND XIO B3:10/8 OTL B3:10/8 EOR
%   B3:10/4  "Press_pack_detected" %
%   B3:10/2  "Press_down_done" %
%   B3:10/3  "Timeout_press_down" %
%   B3:2/2  B62  "B62-Sensor check flap" %
%   B3:0/3  B10  "DETECTION HEAD PACK" %
%   B3:10/8  "Press_down_check_fla p1" %

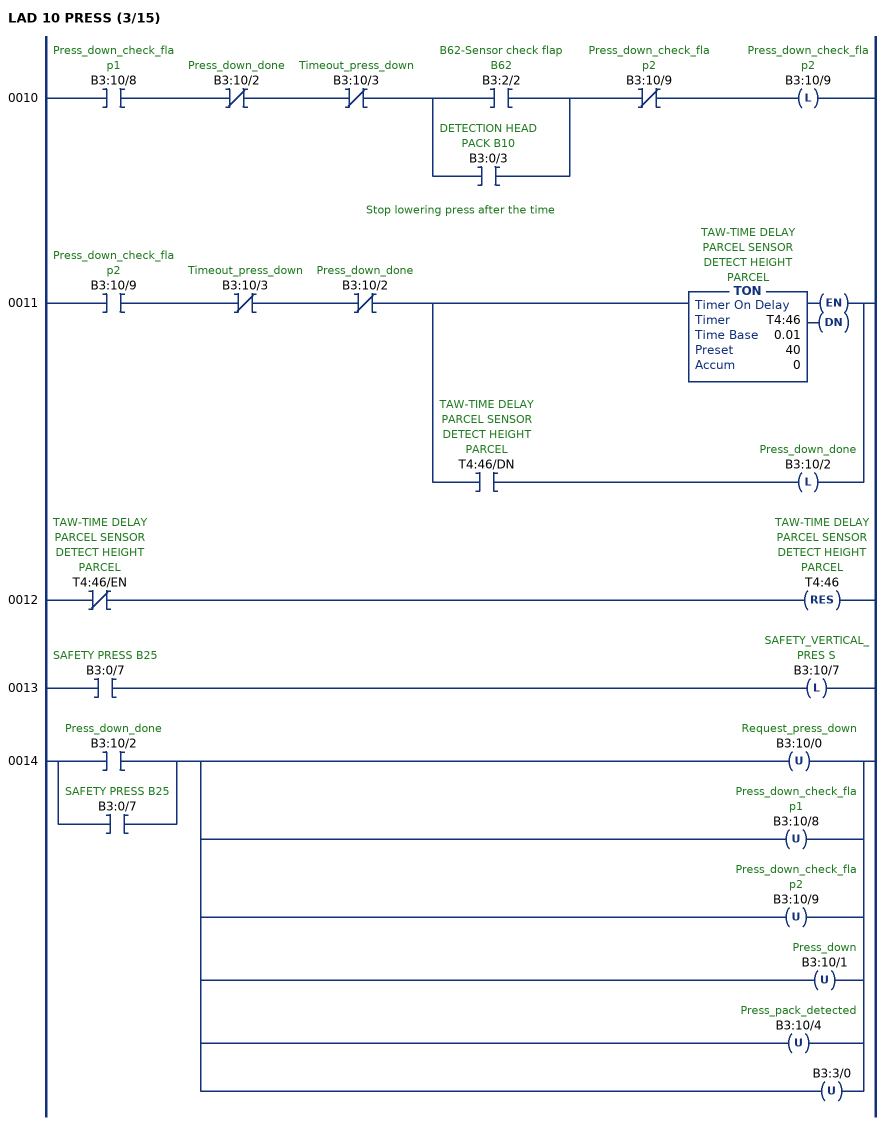
% Rung: 10 %
SOR XIC B3:10/8 XIO B3:10/2 XIO B3:10/3 BST XIC B3:2/2 NXB XIC B3:0/3 BND XIO B3:10/9 OTL B3:10/9 EOR
%   B3:10/8  "Press_down_check_fla p1" %
%   B3:10/2  "Press_down_done" %
%   B3:10/3  "Timeout_press_down" %
%   B3:2/2  B62  "B62-Sensor check flap" %
%   B3:0/3  B10  "DETECTION HEAD PACK" %
%   B3:10/9  "Press_down_check_fla p2" %
% Rung: 11 %
% Stop lowering press after the time %
SOR XIC B3:10/9 XIO B3:10/3 XIO B3:10/2 BST TON T4:46 0.01 40 0 NXB XIC T4:46/DN OTL B3:10/2 BND EOR
%   B3:10/9  "Press_down_check_fla p2" %
%   B3:10/3  "Timeout_press_down" %
%   B3:10/2  "Press_down_done" %
%   T4:46  "TAW-TIME DELAY PARCEL SENSOR DETECT HEIGHT PARCEL" %
% Rung: 12 %
SOR XIO T4:46/EN RES T4:46 EOR
%   T4:46  "TAW-TIME DELAY PARCEL SENSOR DETECT HEIGHT PARCEL" %
% Rung: 13 %
SOR XIC B3:0/7 OTL B3:10/7 EOR
%   B3:0/7  B25  "SAFETY PRESS" %
%   B3:10/7  "SAFETY_VERTICAL_PRES S" %
% Rung: 14 %
SOR BST XIC B3:10/2 NXB XIC B3:0/7 BND BST BST BST OTU B3:10/0 NXB BST OTU B3:10/8 NXB OTU B3:10/9 BND BND NXB OTU B3:10/1 BND NXB BST OTU B3:10/4 NXB OTU B3:3/0 BND BND EOR
%   B3:10/2  "Press_down_done" %
%   B3:0/7  B25  "SAFETY PRESS" %
%   B3:10/0  "Request_press_down" %
%   B3:10/8  "Press_down_check_fla p1" %
%   B3:10/9  "Press_down_check_fla p2" %
%   B3:10/1  "Press_down" %
%   B3:10/4  "Press_pack_detected" %

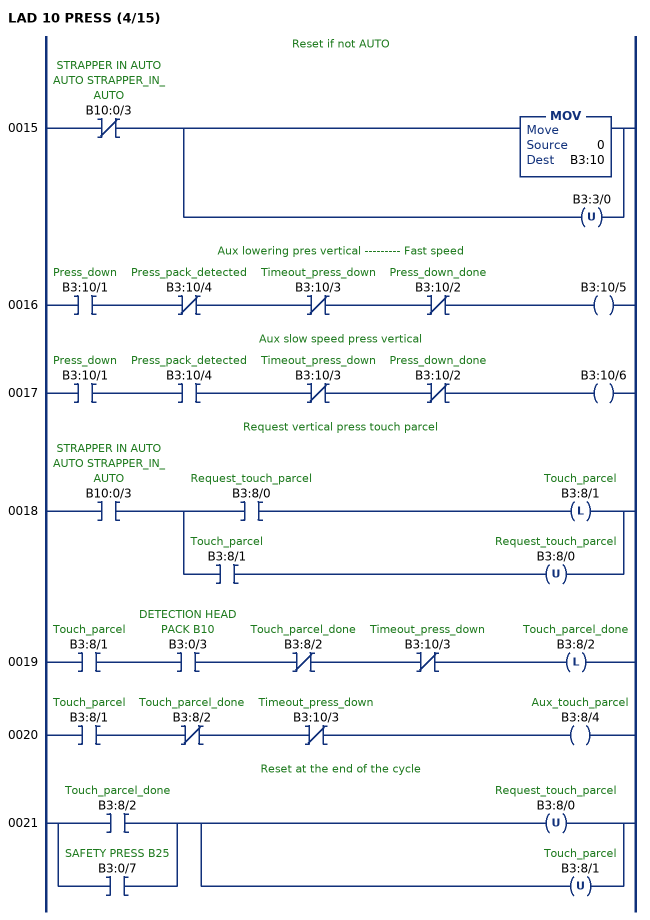
% Rung: 15 %
% Reset if not AUTO %
SOR XIO B10:0/3 BST MOV 0 B3:10 NXB OTU B3:3/0 BND EOR
%   B10:0/3  STRAPPER_IN_AUTO  "STRAPPER IN AUTO AUTO" %
% Rung: 16 %
% Aux lowering pres vertical --------- Fast speed %
SOR XIC B3:10/1 XIO B3:10/4 XIO B3:10/3 XIO B3:10/2 OTE B3:10/5 EOR
%   B3:10/1  "Press_down" %
%   B3:10/4  "Press_pack_detected" %
%   B3:10/3  "Timeout_press_down" %
%   B3:10/2  "Press_down_done" %
% Rung: 17 %
% Aux slow speed press vertical %
SOR XIC B3:10/1 XIC B3:10/4 XIO B3:10/3 XIO B3:10/2 OTE B3:10/6 EOR
%   B3:10/1  "Press_down" %
%   B3:10/4  "Press_pack_detected" %
%   B3:10/3  "Timeout_press_down" %
%   B3:10/2  "Press_down_done" %
% Rung: 18 %
% Request vertical press touch parcel %
SOR XIC B10:0/3 BST XIC B3:8/0 OTL B3:8/1 NXB XIC B3:8/1 OTU B3:8/0 BND EOR
%   B10:0/3  STRAPPER_IN_AUTO  "STRAPPER IN AUTO AUTO" %
%   B3:8/0  "Request_touch_parcel" %
%   B3:8/1  "Touch_parcel" %
% Rung: 19 %
SOR XIC B3:8/1 XIC B3:0/3 XIO B3:8/2 XIO B3:10/3 OTL B3:8/2 EOR
%   B3:8/1  "Touch_parcel" %
%   B3:0/3  B10  "DETECTION HEAD PACK" %
%   B3:8/2  "Touch_parcel_done" %
%   B3:10/3  "Timeout_press_down" %
% Rung: 20 %
SOR XIC B3:8/1 XIO B3:8/2 XIO B3:10/3 OTE B3:8/4 EOR
%   B3:8/1  "Touch_parcel" %
%   B3:8/2  "Touch_parcel_done" %
%   B3:10/3  "Timeout_press_down" %
%   B3:8/4  "Aux_touch_parcel" %
% Rung: 21 %
% Reset at the end of the cycle %
SOR BST XIC B3:8/2 NXB XIC B3:0/7 BND BST OTU B3:8/0 NXB OTU B3:8/1 BND EOR
%   B3:8/2  "Touch_parcel_done" %
%   B3:0/7  B25  "SAFETY PRESS" %
%   B3:8/0  "Request_touch_parcel" %
%   B3:8/1  "Touch_parcel" %

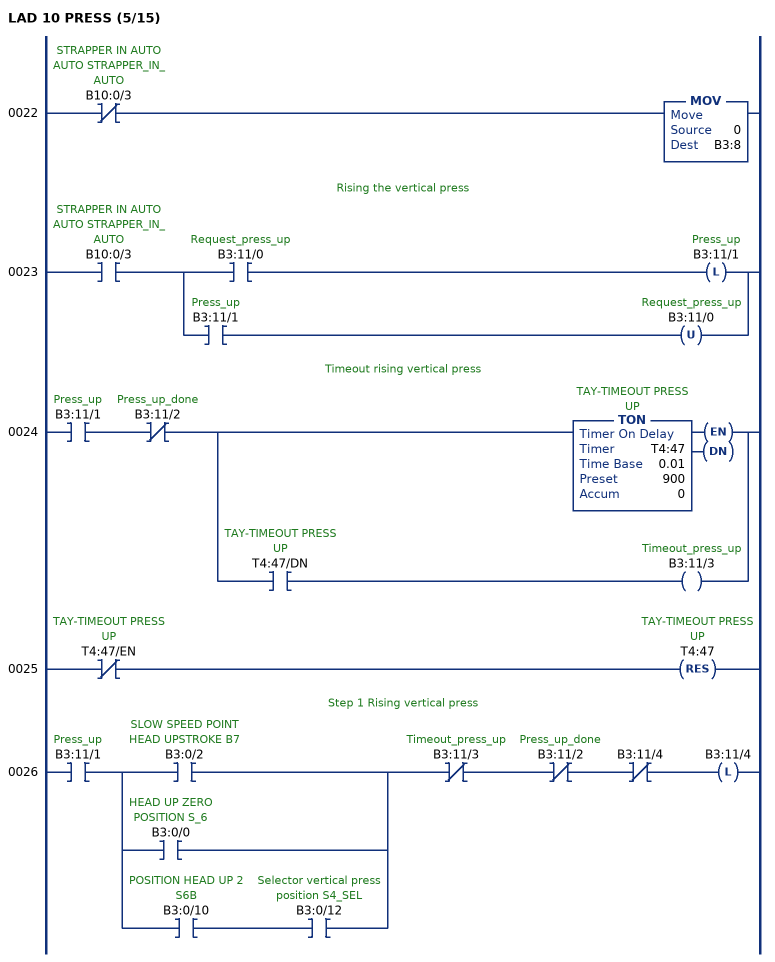
% Rung: 22 %
SOR XIO B10:0/3 MOV 0 B3:8 EOR
%   B10:0/3  STRAPPER_IN_AUTO  "STRAPPER IN AUTO AUTO" %
% Rung: 23 %
% Rising the vertical press %
SOR XIC B10:0/3 BST XIC B3:11/0 OTL B3:11/1 NXB XIC B3:11/1 OTU B3:11/0 BND EOR
%   B10:0/3  STRAPPER_IN_AUTO  "STRAPPER IN AUTO AUTO" %
%   B3:11/0  "Request_press_up" %
%   B3:11/1  "Press_up" %
% Rung: 24 %
% Timeout rising vertical press %
SOR XIC B3:11/1 XIO B3:11/2 BST TON T4:47 0.01 900 0 NXB XIC T4:47/DN OTE B3:11/3 BND EOR
%   B3:11/1  "Press_up" %
%   B3:11/2  "Press_up_done" %
%   T4:47  "TAY-TIMEOUT PRESS UP" %
%   B3:11/3  "Timeout_press_up" %
% Rung: 25 %
SOR XIO T4:47/EN RES T4:47 EOR
%   T4:47  "TAY-TIMEOUT PRESS UP" %
% Rung: 26 %
% Step 1 Rising vertical press %
SOR XIC B3:11/1 BST XIC B3:0/2 NXB BST XIC B3:0/0 NXB XIC B3:0/10 XIC B3:0/12 BND BND XIO B3:11/3 XIO B3:11/2 XIO B3:11/4 OTL B3:11/4 EOR
%   B3:11/1  "Press_up" %
%   B3:0/2  B7  "SLOW SPEED POINT HEAD UPSTROKE" %
%   B3:0/0  S_6  "HEAD UP ZERO POSITION" %
%   B3:0/10  S6B  "POSITION HEAD UP 2" %
%   B3:0/12  S4_SEL  "Selector vertical press position" %
%   B3:11/3  "Timeout_press_up" %
%   B3:11/2  "Press_up_done" %

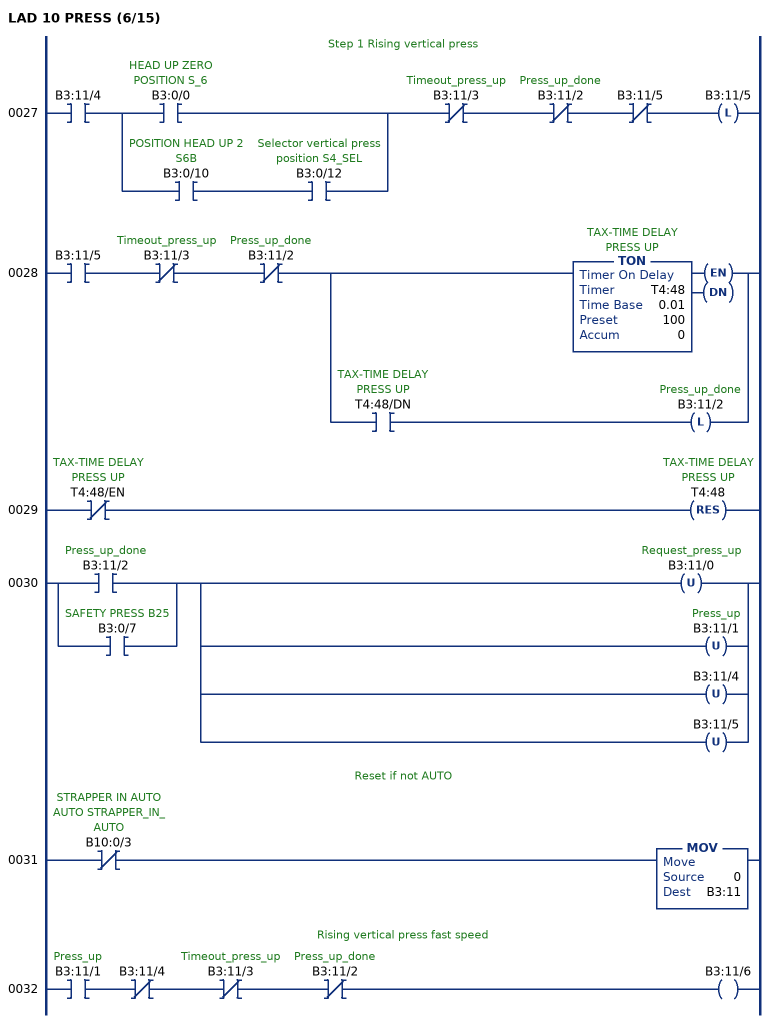
% Rung: 27 %
% Step 1 Rising vertical press %
SOR XIC B3:11/4 BST XIC B3:0/0 NXB XIC B3:0/10 XIC B3:0/12 BND XIO B3:11/3 XIO B3:11/2 XIO B3:11/5 OTL B3:11/5 EOR
%   B3:0/0  S_6  "HEAD UP ZERO POSITION" %
%   B3:0/10  S6B  "POSITION HEAD UP 2" %
%   B3:0/12  S4_SEL  "Selector vertical press position" %
%   B3:11/3  "Timeout_press_up" %
%   B3:11/2  "Press_up_done" %
% Rung: 28 %
SOR XIC B3:11/5 XIO B3:11/3 XIO B3:11/2 BST TON T4:48 0.01 100 0 NXB XIC T4:48/DN OTL B3:11/2 BND EOR
%   B3:11/3  "Timeout_press_up" %
%   B3:11/2  "Press_up_done" %
%   T4:48  "TAX-TIME DELAY PRESS UP" %
% Rung: 29 %
SOR XIO T4:48/EN RES T4:48 EOR
%   T4:48  "TAX-TIME DELAY PRESS UP" %
% Rung: 30 %
SOR BST XIC B3:11/2 NXB XIC B3:0/7 BND BST BST OTU B3:11/0 NXB OTU B3:11/1 BND NXB BST OTU B3:11/4 NXB OTU B3:11/5 BND BND EOR
%   B3:11/2  "Press_up_done" %
%   B3:0/7  B25  "SAFETY PRESS" %
%   B3:11/0  "Request_press_up" %
%   B3:11/1  "Press_up" %
% Rung: 31 %
% Reset if not AUTO %
SOR XIO B10:0/3 MOV 0 B3:11 EOR
%   B10:0/3  STRAPPER_IN_AUTO  "STRAPPER IN AUTO AUTO" %
% Rung: 32 %
% Rising vertical press fast speed %
SOR XIC B3:11/1 XIO B3:11/4 XIO B3:11/3 XIO B3:11/2 OTE B3:11/6 EOR
%   B3:11/1  "Press_up" %
%   B3:11/3  "Timeout_press_up" %
%   B3:11/2  "Press_up_done" %

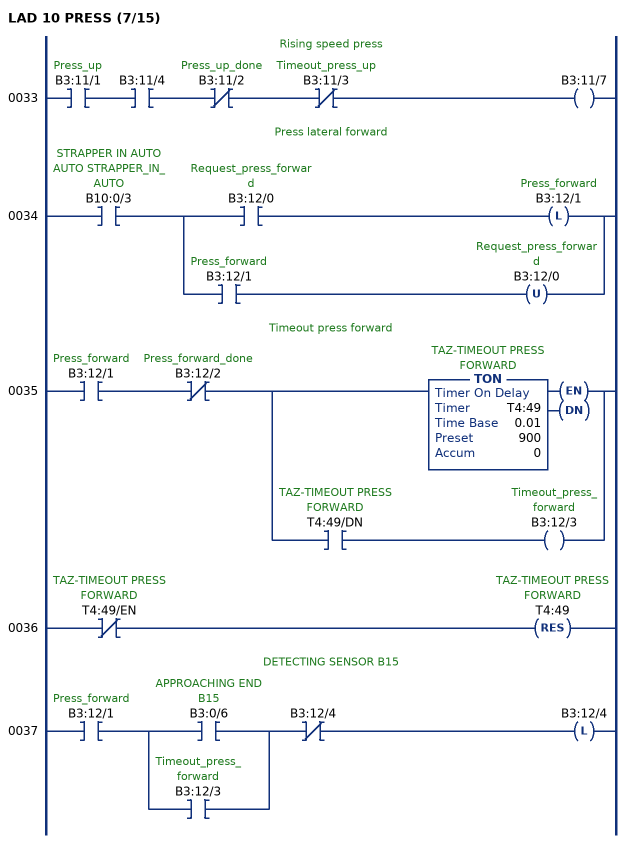
% Rung: 33 %
% Rising speed press %
SOR XIC B3:11/1 XIC B3:11/4 XIO B3:11/2 XIO B3:11/3 OTE B3:11/7 EOR
%   B3:11/1  "Press_up" %
%   B3:11/2  "Press_up_done" %
%   B3:11/3  "Timeout_press_up" %
% Rung: 34 %
% Press lateral forward %
SOR XIC B10:0/3 BST XIC B3:12/0 OTL B3:12/1 NXB XIC B3:12/1 OTU B3:12/0 BND EOR
%   B10:0/3  STRAPPER_IN_AUTO  "STRAPPER IN AUTO AUTO" %
%   B3:12/0  "Request_press_forwar d" %
%   B3:12/1  "Press_forward" %
% Rung: 35 %
% Timeout press forward %
SOR XIC B3:12/1 XIO B3:12/2 BST TON T4:49 0.01 900 0 NXB XIC T4:49/DN OTE B3:12/3 BND EOR
%   B3:12/1  "Press_forward" %
%   B3:12/2  "Press_forward_done" %
%   T4:49  "TAZ-TIMEOUT PRESS FORWARD" %
%   B3:12/3  "Timeout_press_ forward" %
% Rung: 36 %
SOR XIO T4:49/EN RES T4:49 EOR
%   T4:49  "TAZ-TIMEOUT PRESS FORWARD" %
% Rung: 37 %
% DETECTING SENSOR B15 %
SOR XIC B3:12/1 BST XIC B3:0/6 NXB XIC B3:12/3 BND XIO B3:12/4 OTL B3:12/4 EOR
%   B3:12/1  "Press_forward" %
%   B3:0/6  B15  "APPROACHING END" %
%   B3:12/3  "Timeout_press_ forward" %

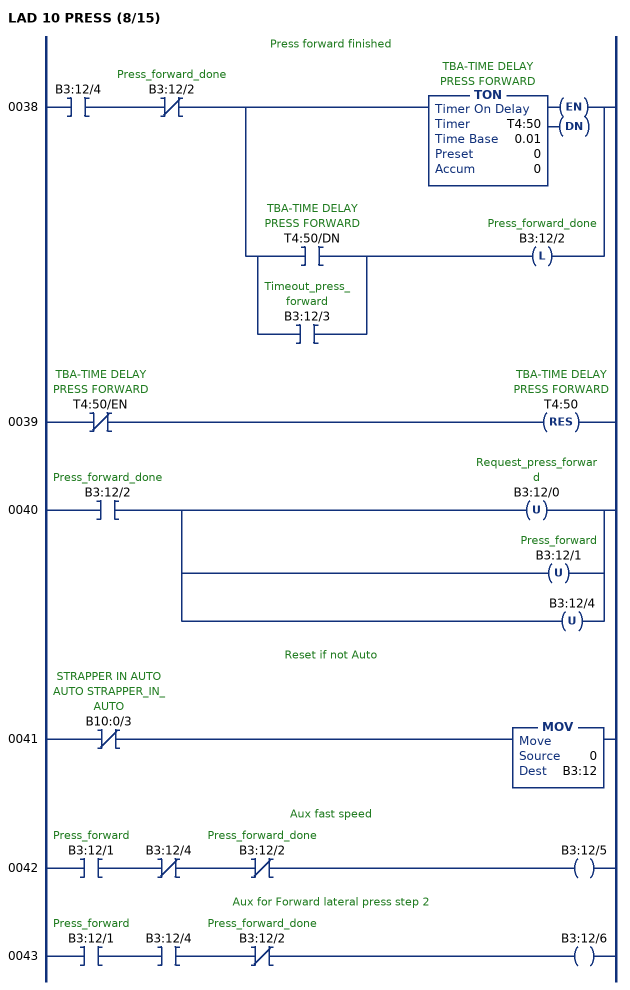
% Rung: 38 %
% Press forward finished %
SOR XIC B3:12/4 XIO B3:12/2 BST TON T4:50 0.01 0 0 NXB BST XIC T4:50/DN NXB XIC B3:12/3 BND OTL B3:12/2 BND EOR
%   B3:12/2  "Press_forward_done" %
%   T4:50  "TBA-TIME DELAY PRESS FORWARD" %
%   B3:12/3  "Timeout_press_ forward" %
% Rung: 39 %
SOR XIO T4:50/EN RES T4:50 EOR
%   T4:50  "TBA-TIME DELAY PRESS FORWARD" %
% Rung: 40 %
SOR XIC B3:12/2 BST BST OTU B3:12/0 NXB OTU B3:12/1 BND NXB OTU B3:12/4 BND EOR
%   B3:12/2  "Press_forward_done" %
%   B3:12/0  "Request_press_forwar d" %
%   B3:12/1  "Press_forward" %
% Rung: 41 %
% Reset if not Auto %
SOR XIO B10:0/3 MOV 0 B3:12 EOR
%   B10:0/3  STRAPPER_IN_AUTO  "STRAPPER IN AUTO AUTO" %
% Rung: 42 %
% Aux fast speed %
SOR XIC B3:12/1 XIO B3:12/4 XIO B3:12/2 OTE B3:12/5 EOR
%   B3:12/1  "Press_forward" %
%   B3:12/2  "Press_forward_done" %
% Rung: 43 %
% Aux for Forward lateral press step 2 %
SOR XIC B3:12/1 XIC B3:12/4 XIO B3:12/2 OTE B3:12/6 EOR
%   B3:12/1  "Press_forward" %
%   B3:12/2  "Press_forward_done" %

